(* CODESYS project CDPR_4cables.library
   Title: CDPR_4cables_kinematics_library
   Version: 1.0
   Placeholder: CDPR_4cables_kinematics_library
   Company: EN.EDI research group

Project tree, tasks and I/O mapping:
  libraries: Tc2_Math, * (Beckhoff Automation GmbH); Tc2_Standard, * (Beckhoff Automation GmbH); Tc2_System, * (Beckhoff Automation GmbH); Tc2_Utilities, * (Beckhoff Automation GmbH); Tc3_Module, * (Beckhoff Automation GmbH)
  DUTs/
    data type Eq2order
    data type EqSphere
    data type Matrix2D
    data type Plane
    data type Pose3D
    data type Sphere
    data type WorkspaceLimits
  GVLs/
  POUs/
    FwKinematics_Functions/
      function GetLineSphereIntersection [ST]
      function GetMutualPoint [ST]
      function GetNormalVector [ST]
      function GetSphereEq [ST]
      function GetSphereFromEquation [ST]
      function GetSphereIntersection [ST]
    Kinematics/
      function InvKin_4cables [ST]
      function DirKin_4cables_Sphere [ST]
      function DirKin_4cables_NR [ST]
    Matrix/
      function GetDeterminant2D [ST]
      function GetDeterminant3D [ST]
      function GetInverseMatrix2D [ST]
      function GetVectorialProduct [ST]
      function LU_Decomposition [ST]
      function LU_Factorization [ST]
      function Multiply2DMatrix [ST]
      function SetMatrix2D [ST]
    Other/
      function CheckWorkspace [ST]
      function GetMvectors [ST]
      function GetQvectors [ST]
      function SolveEq2Order [ST]
  VISUs/
*)

// DUTs/Eq2order
//Second order equation=> x2*x^2+x1*x+d=0
TYPE Eq2order :
STRUCT
	x2:LREAL;
	x1:LREAL;
	d:LREAL;
END_STRUCT
END_TYPE

// DUTs/EqSphere
//Sphere equation => x^2+Ax+y^2+By+z^2+Cz+D=0

TYPE EqSphere :
STRUCT
	a: LREAL;	//a is the factor multiplying X
	b: LREAL;	//b is the factor multiplying Y
	c: LREAL;	//c is the factor multiplying Z
	d: LREAL;	//d is the contribution of each coordinate of the center X,Y,Z and the radius
END_STRUCT
END_TYPE

// DUTs/Matrix2D
(*
Matrix:= [
			A	C
			B	D
					]
*)
TYPE Matrix2D :
STRUCT
	A:LREAL;
	B:LREAL;
	C:LREAL;
	D:LREAL;
END_STRUCT
END_TYPE

// DUTs/Plane
//Plane equation=> Ax+By+Cz+D=0
TYPE Plane :
STRUCT
	A: LREAL;
	B: LREAL;
	C: LREAL;
	D: LREAL;
END_STRUCT
END_TYPE

// DUTs/Pose3D
TYPE Pose3D :
STRUCT
	x: LREAL;
	y: LREAL;
	z: LREAL;
	a: LREAL; // if -9999, error
END_STRUCT
END_TYPE

// DUTs/Sphere
//Sphere equation (2)=>

TYPE Sphere :
STRUCT
	x: LREAL;
	y: LREAL;
	z: LREAL;
	radius: LREAL;
END_STRUCT
END_TYPE

// DUTs/WorkspaceLimits
TYPE WorkspaceLimits :
STRUCT
	LimitX_neg:LREAL;
	LimitX_pos:LREAL;
	LimitY_neg:LREAL;
	LimitY_pos:LREAL;
	LimitZ_neg:LREAL;
	LimitZ_pos:LREAL;
END_STRUCT
END_TYPE

// POUs/FwKinematics_Functions/GetLineSphereIntersection
FUNCTION GetLineSphereIntersection : ARRAY[1..2] OF Pose3D
VAR_INPUT
	sphereEquation: EqSphere;
	pv:  Pose3D; 	//parallel_vector
	mp0: Pose3D;	//mutual_point0
END_VAR
VAR
	sphere: Sphere;
	eqLineInSphere:Eq2order;
	t: ARRAY[1..2] OF LREAL;
	ptoSol: ARRAY[1..2] OF Pose3D;
	i: UINT;
END_VAR

//Intersection line-sphere (substitution of line (x,y,z) into sphere)
// line = pv*t + mp0 (equation of line)
sphere:=GetSphereFromEquation(sphereEquation);

eqLineInSphere.x2:=LREAL_TO_REAL(EXPT(pv.x,2)+EXPT(pv.y,2)+EXPT(pv.z,2));
eqLineInSphere.x1:=LREAL_TO_REAL(2*pv.x*(mp0.x-sphere.x)+2*pv.y*(mp0.y-sphere.y)+2*pv.z*(mp0.z-sphere.z));
eqLineInSphere.d:=EXPT(sphere.x,2)+EXPT(sphere.y,2)+EXPT(sphere.z,2)+EXPT(mp0.x,2)+EXPT(mp0.y,2)+EXPT(mp0.z,2)
-2*(sphere.x*mp0.x+sphere.y*mp0.y+sphere.z*mp0.z)-EXPT(sphere.radius,2);

t:=SolveEq2Order(eqLineInSphere.x2,eqLineInSphere.x1,eqLineInSphere.d);

FOR i:=1 TO 2 DO 
	ptoSol[i].x:=pv.x*t[i]+mp0.x;
	ptoSol[i].y:=pv.y*t[i]+mp0.y;
	ptoSol[i].z:=pv.z*t[i]+mp0.z;
END_FOR

GetLineSphereIntersection:=ptoSol;

END_FUNCTION

// POUs/FwKinematics_Functions/GetSphereFromEquation
FUNCTION GetSphereFromEquation : Sphere
VAR_INPUT
	sphereEquation: EqSphere;
END_VAR
VAR
	sphereSol: Sphere;
END_VAR

sphereSol.x:= -sphereEquation.A/2;
sphereSol.y:= -sphereEquation.B/2;
sphereSol.z:= -sphereEquation.C/2;
sphereSol.radius:=SQRT(EXPT(sphereSol.x,2)+EXPT(sphereSol.y,2)+EXPT(sphereSol.z,2)-sphereEquation.d);

GetSphereFromEquation:=sphereSol;

END_FUNCTION

// POUs/Other/SolveEq2Order
FUNCTION SolveEq2Order : ARRAY[1..2] OF LREAL
VAR_INPUT
	x2,x,d:LREAL;
END_VAR
VAR
	a,b,c:LREAL;
	sol:ARRAY[1..2] OF LREAL;
	discriminant: LREAL;
END_VAR

a:=x2;
b:=x;
c:=d;
sol[1]:=0;
sol[2]:=0;

discriminant:=b*b-4*a*c;

IF discriminant < 0 THEN
	sol[1]:=0;
	sol[2]:=0;
END_IF
IF discriminant = 0 THEN
	sol[1]:=-b/(2*a);
	sol[2]:=sol[1];
END_IF
IF discriminant > 0 THEN
	sol[1]:=(-b+SQRT(discriminant))/(2*a);
	sol[2]:=(-b-SQRT(discriminant))/(2*a);
END_IF

SolveEq2Order:=sol;

END_FUNCTION

// POUs/FwKinematics_Functions/GetMutualPoint
FUNCTION GetMutualPoint : Pose3D
VAR_INPUT
	planeA: Plane;
	planeB: Plane;
END_VAR
VAR
	mA: Matrix2D;
	mB: Matrix2D;
	invA: Matrix2D;
	mSol: Matrix2D;
	pSol: Pose3D;
	opc: UINT:=0;
END_VAR

(* Selection of the fixed parameter to obtain the other two variables *)
IF planeA.C=0 AND planeB.C=0 THEN
	opc:=1;
END_IF

IF planeA.B=0 AND planeB.B=0 THEN
	opc:=2;
END_IF

IF planeA.A=0 AND planeB.A=0 THEN
	opc:=3;
END_IF

CASE opc OF
	1:	//X-Y   Z-fixed
		mA.A:=planeA.A;
		mA.B:=planeA.B;
		mA.C:=planeB.A;
		mA.D:=planeB.B;
	2:	//X-Z   Y-fixed
		mA.A:=planeA.A;
		mA.B:=planeA.C;
		mA.C:=planeB.A;
		mA.D:=planeB.C;
	3:	//Y-Z   X-fixed
		mA.A:=planeA.B;
		mA.B:=planeA.C;
		mA.C:=planeB.B;
		mA.D:=planeB.C;
END_CASE

invA:=GetInverseMatrix2D(mA);
		
//We ignore B and D because we want only the first column (matrix 2x1).
//Addd the minus sign because we change the side of the equation
//If the plane is Ax+By+Cz+D=0, we pass to Ax+By+Cz=-D
 
mB.A:=-planeA.D;
mB.B:=0; 
mB.C:=-planeB.D;
mB.D:=0;
mSol:=Multiply2DMatrix(invA, mB);

CASE opc OF
	1: //X-Y
		pSol.x:=mSol.A;
		pSol.y:=mSol.C;	
	2: //X-Z
		pSol.x:=mSol.A;
		pSol.z:=mSol.C;	
	3: //Y-Z
		pSol.y:=mSol.A;
		pSol.Z:=mSol.C;	
END_CASE
		
GetMutualPoint:=pSol;

END_FUNCTION

// POUs/Matrix/GetInverseMatrix2D
FUNCTION GetInverseMatrix2D : Matrix2D
VAR_INPUT
	matrix: Matrix2D;
END_VAR
VAR
	adj: Matrix2D;
	det: LREAL;
	inverse: Matrix2D;
END_VAR

det:=GetDeterminant2D(matrix);

adj:=SetMatrix2D(matrix.D, -matrix.B, -matrix.C, matrix.A);

IF det <> 0 THEN
	inverse.A:=adj.A/det;
	inverse.B:=adj.B/det;
	inverse.C:=adj.C/det;
	inverse.D:=adj.D/det;
ELSE	//ERROR
	inverse.A:=-9999;
	inverse.B:=-9999;
	inverse.C:=-9999;
	inverse.D:=-9999;
END_IF

GetInverseMatrix2D:=inverse;

END_FUNCTION

// POUs/Matrix/GetDeterminant2D
FUNCTION GetDeterminant2D : LREAL
VAR_INPUT
	matrix: Matrix2D;
END_VAR
VAR
	det: LREAL;
END_VAR

det:=Matrix.A*matrix.D-matrix.B*matrix.C;

GetDeterminant2D:=det;

END_FUNCTION

// POUs/Matrix/SetMatrix2D
FUNCTION SetMatrix2D : Matrix2D
VAR_INPUT
	A,B,C,D: LREAL;
END_VAR
VAR
	matrix:Matrix2D;
END_VAR

matrix.A:=A;
matrix.B:=B;
matrix.C:=C;
matrix.D:=D;

SetMatrix2D:=Matrix;

END_FUNCTION

// POUs/Matrix/Multiply2DMatrix
FUNCTION Multiply2DMatrix : Matrix2D
VAR_INPUT
	m1:Matrix2D;
	m2:Matrix2D;
END_VAR
VAR
	mSol:Matrix2D;
END_VAR

mSol.A:=m1.A*m2.A+m1.B*m2.C;
mSol.B:=m1.A*m2.B+m1.B*m2.D;
mSol.C:=m1.C*m2.A+m1.D*m2.C;
mSol.D:=m1.C*m2.B+m1.D*m2.D;

Multiply2DMatrix:=mSol;

END_FUNCTION

// POUs/FwKinematics_Functions/GetNormalVector
FUNCTION GetNormalVector : Pose3D
VAR_INPUT
	Plane: Plane;
END_VAR
VAR
	n: Pose3D;
END_VAR

n.x:=Plane.A;
n.y:=Plane.B;
n.z:=Plane.C;

GetNormalVector:=n;

END_FUNCTION

// POUs/FwKinematics_Functions/GetSphereEq
FUNCTION GetSphereEq : EqSphere
VAR_INPUT
	Lcable:REAL;
	q: Pose3D;
	m: Pose3D;
END_VAR
VAR
	sphere: EqSphere;
END_VAR

// X, Y, Z, -R
// Disregard the weightings of x^2, y^2, z^2 since the objective is to subtract between spheres, so they cancel each other out.
sphere.a:= +(- 2*m.x)+2*q.x;
sphere.b:=+(- 2*m.y)+ 2*q.y;
sphere.c:=+(-2*m.z)+2*q.z;
sphere.d:=LREAL_TO_REAL((-EXPT(Lcable,2)
					+EXPT(m.x,2)-2*m.x*q.x
					+EXPT(m.y,2)-2*m.y*q.y
					+EXPT(m.z,2)-2*m.z*q.z
					+EXPT(q.x,2)+EXPT(q.y,2)+EXPT(q.z,2)));

GetSphereEq:=sphere;

END_FUNCTION

// POUs/FwKinematics_Functions/GetSphereIntersection
FUNCTION GetSphereIntersection : Plane
VAR_INPUT
	sphereA: EqSphere;
	sphereB: EqSphere;
END_VAR
VAR
	plane: Plane;
END_VAR

plane.A:= sphereA.a-sphereB.a;
plane.B:= sphereA.b-sphereB.b;
plane.C:= sphereA.c-sphereB.c;
plane.D:=sphereA.d-sphereB.d;

GetSphereIntersection:=plane;

END_FUNCTION

// POUs/Kinematics/InvKin_4cables
FUNCTION InvKin_4cables : ARRAY[1..4] OF REAL
VAR_INPUT
	q: ARRAY[1..4] OF Pose3D;
	m: ARRAY[1..4] OF Pose3D;
	pObj: Pose3D;	//Spatial objective point to be converted to lengths
END_VAR
VAR
	Li: ARRAY[0..3] OF REAL;
	lengths: ARRAY[0..3] OF REAL;
	i: INT;
END_VAR

FOR i:=1 TO 4 DO
	//Computation of the length vectors
	Li[i-1]:=EXPT(q[i].x+pObj.x-m[i].x,2)+EXPT(q[i].y+pObj.y-m[i].y,2)+EXPT(q[i].z+pObj.z-m[i].z,2);
	lengths[i-1]:=SQRT(Li[i-1]);
END_FOR

InvKin_4cables:=lengths;

END_FUNCTION

// POUs/Kinematics/DirKin_4cables_Sphere
FUNCTION DirKin_4cables_Sphere : Pose3D
VAR_INPUT
	q: ARRAY[1..4]OF Pose3D;
	m: ARRAY[1..4]OF Pose3D;
	l: ARRAY[1..4] OF REAL;
	wp: WorkspaceLimits;
END_VAR
VAR
	sphereEq1: EqSphere;
	sphereEq2: EqSphere;
	sphereEq3: EqSphere;
	plane12: Plane;
	plane13: Plane;
	n12: Pose3D;
	n13: Pose3D;
	u: Pose3D;
	mA: Matrix2D;
	mB: Matrix2D;
	msol: Matrix2D;
	p0: Pose3D;
	ptoSol: ARRAY[1..2] OF Pose3D;		//Two posible solution of the direct kinematics
	fwPtoSol: Pose3D;					//Point solution of the direct kinematics
END_VAR

sphereEq1:=GetSphereEq(q:=q[1],m:=m[1],Lcable:=l[1]);
sphereEq2:=GetSphereEq(q:=q[2],m:=m[2],Lcable:=l[2]);
sphereEq3:=GetSphereEq(q:=q[3],m:=m[3],Lcable:=l[3]);

plane12:=GetSphereIntersection(sphereEq1,sphereEq2);
plane13:=GetSphereIntersection(sphereEq1,sphereEq3);

p0:=GetMutualPoint(plane12,plane13);

n12:=GetNormalVector(plane12);
n13:=GetNormalVector(plane13);

u:=GetVectorialProduct(n12,n13);

ptoSol:=GetLineSphereIntersection(sphereEquation:=sphereEq1,pv:=u,mp0:=p0);

IF checkworkspace(wp:=wp,point:=ptoSol[1]) THEN
	fwPtoSol:=ptoSol[1];
END_IF

IF checkworkspace(wp:=wp,point:=ptoSol[2]) THEN
	fwPtoSol:=ptoSol[2];
END_IF

DirKin_4cables_Sphere:=fwPtoSol;

END_FUNCTION

// POUs/Matrix/GetVectorialProduct
FUNCTION GetVectorialProduct : Pose3D
VAR_INPUT
	v1: Pose3D;
	v2: Pose3D;
END_VAR
VAR
	sol: Pose3D;
END_VAR

sol.x:=v1.y*v2.z-v1.z*v2.y;
sol.y:=v1.z*v2.x-v1.x*v2.z;
sol.z:=v1.x*v2.y-v1.y*v2.x;

GetVectorialProduct:=sol;

END_FUNCTION

// POUs/Other/CheckWorkspace
FUNCTION CheckWorkspace : BOOL
VAR_INPUT
	wp: WorkspaceLimits;
	point: Pose3D;
END_VAR
VAR
	valid: BOOL;
END_VAR

valid:= FALSE;
IF (wp.LimitX_neg <= point.X AND wp.LimitX_pos>= point.X AND 
	wp.LimitY_neg <= point.y AND wp.LimitY_pos>= point.y AND
	wp.LimitZ_neg <= point.z AND wp.LimitZ_pos >= point.z) THEN
	valid:=TRUE;
END_IF

CheckWorkspace:=valid;

END_FUNCTION

// POUs/Kinematics/DirKin_4cables_NR
FUNCTION DirKin_4cables_NR : Pose3D
VAR_INPUT
	q: ARRAY[1..4] OF Pose3D;
	m: ARRAY[1..4] OF Pose3D;
	l: ARRAY[1..4] OF REAL;
	pIni: Pose3D;				//Initial point for the newton-raphson algorithm
	threshold:REAL:=0.01;
	iterations: INT:=100;		//The value of this parameter can be adjusted according to the cycle time of the PLC and the desired accuracy (threshold).
END_VAR
VAR
	alpha: REAL;
	i,j: INT;
	u: ARRAY[0..3] OF REAL;
	v: ARRAY[0..3] OF REAL;
	w: ARRAY[0..3] OF REAL;
	xi: ARRAY[0..3] OF REAL;
	yi: ARRAY[0..3] OF REAL;
	zi: ARRAY[0..3] OF REAL;
	Li: ARRAY[0..3] OF REAL;
	long: ARRAY[0..3] OF REAL;
	Fi: ARRAY[0..3] OF REAL;
	r11,r12,r13,r21,r22,r23,r31,r32,r33:REAL;
	a:INT;
	Jac1: ARRAY[0..3]OF REAL;
	Jac2: ARRAY[0..3]OF REAL;
	Jac3: ARRAY[0..3]OF REAL;
	Jac4: ARRAY[0..3]OF REAL;
	Jac4D: ARRAY[0..3,0..3] OF REAL;
	Jac3D: ARRAY[0..2,0..2] OF REAL;
	matricesUL:ARRAY[1..2] OF ARRAY[0..3,0..3] OF REAL;
	Uaux:ARRAY[0..3,0..3] OF REAL;
	Laux:ARRAY[0..3,0..3] OF REAL;
	invJac:ARRAY[0..3,0..3] OF REAL;
	sum: ARRAY[0..3] OF REAL;
	newPtoA: Pose3D;
	ptoA:Pose3D;
	diff: ARRAY[0..3] OF REAL;
	k: INT;
	det3D:LREAL;		
	ptoSol: Pose3D;//Point solution of the direct kinematics
END_VAR

ptoA:=pIni;

FOR k:=0 TO iterations DO
	//Initlization of the rotation matrix
	r11:=1;
	r12:=0;
	r13:=0;
	r21:=0;
	r22:=1;
	r23:=0;
	r31:=0;
	r32:=0;
	r33:=1;
	
	FOR i:=1 TO 3 DO
		u[i-1]:=r11*q[i].x+r12*q[i].y+r13*q[i].z;
		v[i-1]:=r21*q[i].x+r22*q[i].y+r23*q[i].z;
		w[i-1]:=r31*q[i].x+r32*q[i].y+r33*q[i].z;
		
		xi[i-1]:=ptoA.x-m[i].x;
		yi[i-1]:=ptoA.y-m[i].y;
		zi[i-1]:=ptoA.z-m[i].z;
		
		//Computation of the length vectors
		Li[i-1]:=EXPT(xi[i-1]+u[i-1],2)+EXPT(yi[i-1]+v[i-1],2)+EXPT(zi[i-1]+w[i-1],2);
		long[i-1]:=SQRT(Li[i-1]);
		
		//Computation of the minimization function (F)
		Fi[i-1]:=Li[i-1]-LREAL_TO_REAL(EXPT(l[i],2));
		
		Jac1[i-1]:=2*(xi[i-1]+u[i-1]);
		Jac2[i-1]:=2*(yi[i-1]+v[i-1]);
		Jac3[i-1]:=2*(zi[i-1]+w[i-1]);
		Jac4[i-1]:=2*(yi[i-1]*u[i-1]-xi[i-1]*v[i-1]);
	END_FOR
	
	FOR i:=0 TO 3 DO
		Jac4D[i,0]:=Jac1[i];
		Jac4D[i,1]:=Jac2[i];
		Jac4D[i,2]:=Jac3[i];
		Jac4D[i,3]:=0;
		
		Jac3D[i,0]:=Jac1[i];
		Jac3D[i,1]:=Jac2[i];
		Jac3D[i,2]:=Jac3[i];
	END_FOR
	
	det3D:=GetDeterminant3D(Jac3D);
	IF (det3D=0) THEN
		newPtoA.a:=-9999;
		DirKin_4cables_NR:=newPtoA;
		EXIT;
	END_IF
	
	//Calculation of the inverse of the Jacobian
	matricesUL:=LU_Decomposition(A:=Jac4D,Indice:=3); //jacobian4D is used with index 3, which disregards the 4th row/column.
	Uaux:=matricesUL[1];
	Laux:=matricesUL[2];
	invJac:=LU_Factorization(L:=Laux,U:=Uaux,Indice:=3); //jacobian4D is used with index 3, which disregards the 4th row/column.
	
	//sum of the multiplication of the inverse of the Jacobian and the F matrix for each direction and orientation component.
	FOR  i:=0 TO 2 BY 1 DO
		sum[i]:=0;
		FOR  j:=0 TO 2 BY 1 DO
			sum[i]:=sum[i]+invJac[i,j]*Fi[j];
		END_FOR;
	END_FOR;
	
	//Calculation of the new iteration point
	newPtoA.x:=ptoA.x-sum[0];
	newPtoA.y:=ptoA.y-sum[1];
	newPtoA.z:=ptoA.z-sum[2];
	
	//Convergence factor calculation
	diff[0]:=ABS(newPtoA.x-ptoA.x);
	diff[1]:=ABS(newPtoA.y-ptoA.y);
	diff[2]:=ABS(newPtoA.z-ptoA.z);
	
	//The convergence factor is checked to determine whether the convergence factor is less than the set precision limit (threshold).
	IF (diff[0]<threshold AND diff[1]<threshold AND diff[2]<threshold) THEN
		DirKin_4cables_NR:=newPtoA;
		EXIT;
	ELSE
		ptoA:=newPtoA;
	END_IF 

END_FOR

END_FUNCTION

// POUs/Matrix/GetDeterminant3D
FUNCTION GetDeterminant3D : LREAL
VAR_INPUT
	m: ARRAY[0..2,0..2] OF REAL;
END_VAR
VAR
END_VAR

GetDeterminant3D:=-(m[0,2]*m[1,1]*m[2,0])+m[0,1]*m[1,2]*m[2,0]+m[0,2]*m[1,0]*m[2,1]-m[0,0]*m[1,2]*m[2,1]-m[0,1]*m[1,0]*m[2,2]+m[0,0]*m[1,1]*m[2,2];

END_FUNCTION

// POUs/Matrix/LU_Decomposition
FUNCTION LU_Decomposition : ARRAY[1..2] OF ARRAY[0..3,0..3] OF REAL
VAR_INPUT
	Indice:INT;
	A: ARRAY[0..3,0..3]OF REAL;
END_VAR
VAR
	U: ARRAY[0..3,0..3] OF REAL;
	L: ARRAY[0..3,0..3] OF REAL;
	i,j,k: INT;
	sum: REAL;
END_VAR

//Initialization of the triangular matrixes 
FOR i := 0 TO (Indice-1) BY 1  DO
	FOR j := 0 TO (Indice-1) BY 1  DO
		L[i,j]:=0;
		U[i,j]:=0;
	END_FOR;
END_FOR;


FOR i := 0 TO (Indice-1) DO
	
	//U matrix
	FOR j := i TO (Indice-1) DO
		
		//Calculation of the sum of element i,j
		sum:=0;
		FOR k := 0 TO i DO
			sum:=sum+(L[i,k]*U[k,j]);
		END_FOR;
		
		//Calculation of the element i,j
		U[i,j]:=A[i,j]-sum;
	END_FOR;
	
	//L-matrix
	FOR j := i TO (Indice-1) DO
		
		//if the next element corresponds to the diagonal of the matrix L...
		IF (i=j) THEN
			L[i,i]:=1;	//Diagonal, it is assigned a '1'.
		ELSE
		
			//Calculation of the sum of element j,i
			sum:=0;
			FOR k := 0 TO i DO
				sum:=sum+(L[j,k]*U[k,i]);
			END_FOR;
			
			//Calculation of the element j,i
			L[j,i]:=(A[j,i]-sum)/U[i,i];
			END_IF;
	END_FOR;
	
END_FOR;

//Assignment of the outputs 
LU_Decomposition[1]:=U;
LU_Decomposition[2]:=L;

END_FUNCTION

// POUs/Matrix/LU_Factorization
FUNCTION LU_Factorization : ARRAY[0..3,0..3]OF REAL
VAR_INPUT
	L: ARRAY[0..3,0..3]OF REAL;
	U: ARRAY[0..3,0..3]OF REAL;
	Indice: INT;
END_VAR
VAR
	matrizI: ARRAY[0..3,0..3] OF REAL;
	Y: ARRAY[0..3,0..3] OF REAL;
	X: ARRAY[0..3,0..3] OF REAL;
	i,j,k: INT;
	sum: REAL;
END_VAR

//Initialization of the matrices
FOR i := 0 TO (Indice-1) BY 1  DO
	FOR j := 0 TO (Indice-1) BY 1  DO
		
		//Initialization of the matrices X and Y
		X[i,j]:=0;
		Y[i,j]:=0;
		
		////Fill I-matrix
		IF (i=j) THEN
			matrizI[i,j]:=1;	//Fill with a '1' the matrix I on its diagonal
		ELSE
			matrizI[i,j]:=0;	//Fill with a '0' in the remaining items
		END_IF;
	END_FOR;
END_FOR;

//Calculation of matrices Y and X
FOR i := 0 TO (Indice-1) DO
	
	//First the Y-matrix calculation is performed.
	FOR j := 0 TO (Indice-1) DO
		
		//The first element of the column is equal to the term of Matrix I (j,i)
		IF (j=0) THEN
			Y[j,i]:=matrizI[j,i];
		ELSE
			
			//Calculating the sum of element i,j
			sum:=0;
			FOR k := 0 TO (j-1) DO
				sum:=sum+L[j,k]*Y[k,i];
			END_FOR;
			
			//Calculation of element j,i
			Y[j,i]:=(matrizI[j,i]-sum)/L[j,j];
		END_IF;
		
	END_FOR;
	
	//X-Matrix
	//First the calculation is performed based on the counter i and the index of the array
	X[(Indice-1),i]:=Y[(Indice-1),i]/U[(Indice-1),(Indice-1)];
	
	//Calculating the remaining elements of X-matrix
	FOR j := (Indice-1)-1 TO 0 BY -1 DO
		
		//Calculating the sum of element i,j
		sum:=0;
		FOR k := j+1 TO (Indice-1) DO
			sum:=sum+U[j,k]*X[k,i];
		END_FOR;
		
		//Calculation of element i,j
		X[j,i]:=(Y[j,i]-sum)/U[j,j];
	END_FOR;
	
END_FOR;

//Assignment of the output matrix (Inverse) with the result of the function
LU_Factorization:=X;

END_FUNCTION

// POUs/Other/GetMvectors
FUNCTION GetMvectors : ARRAY[1..4] OF Pose3D
VAR_INPUT
	Bl:REAL;
	Bh:REAL;
	Bw:REAL;
END_VAR
VAR
	m: ARRAY[1..4]OF Pose3D;
	i: INT;
END_VAR

FOR i:=1 TO 4 DO
	m[i].x:=0;
	m[i].y:=0;
	m[i].z:=0;
END_FOR

m[1].x:=-Bl/2;
m[1].y:=-Bw/2;
m[1].z:=Bh;
m[2].x:=Bl/2;
m[2].y:=-Bw/2;
m[2].z:=Bh;
m[3].x:=Bl/2;
m[3].y:=Bw/2;
m[3].z:=Bh;
m[4].x:=-Bl/2;
m[4].y:=Bw/2;
m[4].z:=Bh;

GetMvectors:=m;

END_FUNCTION

// POUs/Other/GetQvectors
FUNCTION GetQvectors : ARRAY[1..4] OF Pose3D
VAR_INPUT
	Tl:REAL;
	Th:REAL;
	Tw:REAL;
END_VAR
VAR
	q: ARRAY[1..4] OF Pose3D;
	i: INT;
END_VAR

FOR i:=1 TO 4 DO
	q[i].x:=0;
	q[i].y:=0;
	q[i].z:=0;
END_FOR

q[1].x:=-Tl/2;
q[1].y:=-Tw/2;
q[1].z:=Th/2;
q[2].x:=Tl/2;
q[2].y:=-Tw/2;
q[2].z:=Th/2;
q[3].x:=Tl/2;
q[3].y:=Tw/2;
q[3].z:=Th/2;
q[4].x:=-Tl/2;
q[4].y:=Tw/2;
q[4].z:=Th/2;

GetQvectors:=q;

END_FUNCTION
